# EPICS IOC start-up script: calcApp/iocsh/sseq.iocsh
# ### sseq.iocsh ###

#- ###################################################
#- PREFIX         - IOC Prefix
#- INSTANCE       - Instance Prefix
#- CALC           - Location of Calc module
#- ###################################################

#- string sequence (sseq) records
dbLoadRecords("$(CALC)/db/userStringSeqs10.db","P=$(PREFIX)")

#- editSseq - edit any sseq or seq record
dbLoadRecords("$(CALC)/db/editSseq.db", "P=$(PREFIX),Q=$(INSTANCE)")
doAfterIocInit("seq &editSseq, 'P=$(PREFIX),Q=$(INSTANCE)'")
